// TIA Portal V15.1 export
// export: Created 2024-06-21T08:41:25.0501591Z, ExportSetting WithDefaults, DisplayName Totally Integrated Automation Portal, DisplayVersion V15.1 Update 5, DisplayName TIA Portal Openness, DisplayVersion V15.1 Update 5, DisplayName SINAMICS Startdrive Advanced, DisplayVersion V15.1, DisplayName G130, G150, S120, S150, SINAMICS MV, S210, DisplayVersion V15.1, DisplayName G110M, G120, G120C, G120D, G120P, DisplayVersion V15.1, DisplayName STEP 7 Professional, DisplayVersion V15.1 Update 5, DisplayName STEP 7 Safety, DisplayVersion V15.1, DisplayName WinCC Professional, DisplayVersion V15.1 Update 5, DisplayName SIMATIC Visualization Architect, DisplayVersion V15.1
FUNCTION_BLOCK "209230NCB01TagSeq"   // FB440, GRAPH
{ S7_Optimized_Access := 'TRUE' }
VERSION : 0.1
// stored: AcknowledgeErrorsRequired true, AutoNumber false, GraphVersion 6.0, InitialValuesAcquisition false, IsIECCheckEnabled false, LanguageInNetworks FBD, LockOperatingMode false, PermanentILProcessingInMANMode false, SetENOAutomatically false, SkipSteps false, UDAEnableTagReadback false, WithAlarmHandling true
   // inherited from GRAPH_BASE
   VAR
      OFF_SQ_BASE : Bool;
   END_VAR
   VAR_INPUT
      OFF_SQ { ExternalWritable := 'False'} : Bool := false;   // Turn sequence off
      INIT_SQ { ExternalWritable := 'False'} : Bool := false;   // Set sequence to initial state
      ACK_EF { ExternalWritable := 'False'} : Bool := false;   // Acknowledge all errors and faults
      S_PREV { ExternalWritable := 'False'} : Bool := false;   // Output previous step in parameter S_NO
      S_NEXT { ExternalWritable := 'False'} : Bool := false;   // Indicate next step in parameter S_NO
      SW_AUTO { ExternalWritable := 'False'} : Bool := false;   // Automatic mode
      SW_TAP { ExternalWritable := 'False'} : Bool := false;   // Semiautomatic/switch with transition
      SW_TOP { ExternalWritable := 'False'} : Bool := false;   // Semiautomatic/ignore transition
      SW_MAN { ExternalWritable := 'False'} : Bool := false;   // Manual mode
      S_SEL { ExternalWritable := 'False'} : Int := 0;   // Select step to be output to S_NO
      S_ON { ExternalWritable := 'False'} : Bool := false;   // Activate step indicated in S_NO
      S_OFF { ExternalWritable := 'False'} : Bool := false;   // Deactivate step indicated S_NO
      T_PUSH { ExternalWritable := 'False'} : Bool := false;   // Enable transition to switch in semi automatic mode
   END_VAR
   VAR_OUTPUT
      S_NO { ExternalWritable := 'False'} : Int := 0;   // Step number
      S_MORE { ExternalWritable := 'False'} : Bool := false;   // More steps are available and can be shown in S_NO
      S_ACTIVE { ExternalWritable := 'False'} : Bool := false;   // Step indicated in S_NO is active
      ERR_FLT { ExternalWritable := 'False'} : Bool := false;   // Interlock or supervision group error
      AUTO_ON { ExternalWritable := 'False'} : Bool := false;   // Automatic mode is active
      TAP_ON { ExternalWritable := 'False'} : Bool := false;   // Semiautomatic mode/step with transition enabled
      TOP_ON { ExternalWritable := 'False'} : Bool := false;   // Semiautomatic mode/ignore transition enabled
      MAN_ON { ExternalWritable := 'False'} : Bool := false;   // Manual mode is active
   END_VAR
BEGIN
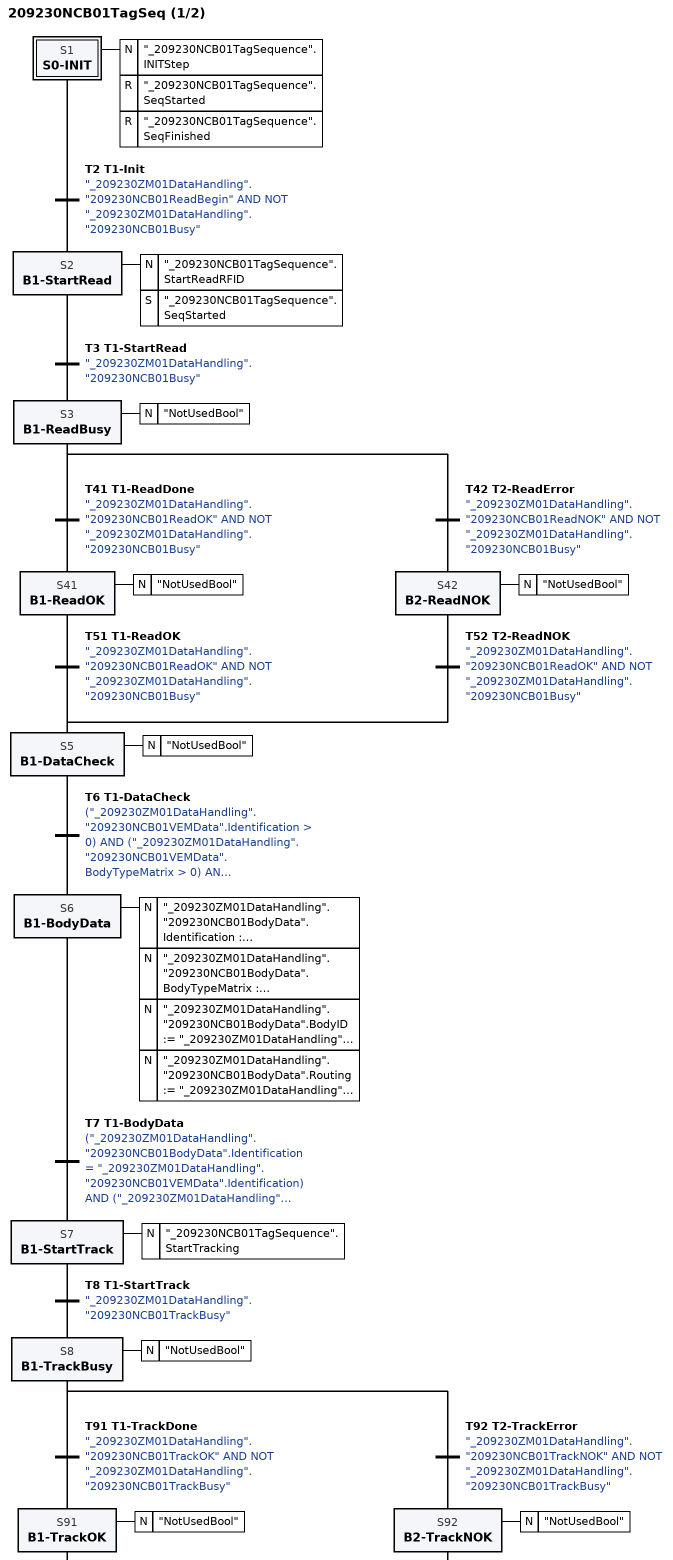
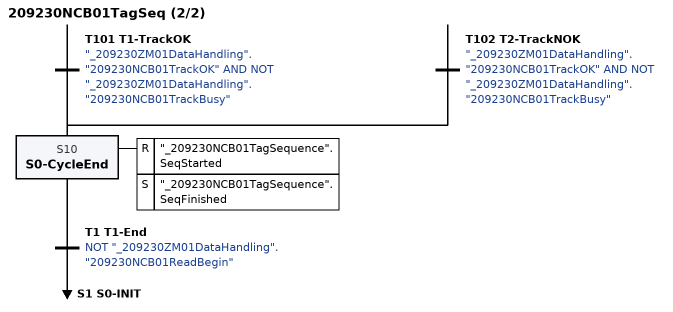
   // sequencer 1: 209230NCB01 Tag Sequence
   // Tag Sequence of 209230NCB01
   INITIAL_STEP "S0-INIT":   // S1, max time T#10S, warning time T#7S
      interlock C := (none);   // Not used
      supervision V := (none);   // Not Used
      // INIT
              N    "_209230NCB01TagSequence".INITStep
              R    "_209230NCB01TagSequence".SeqStarted
              R    "_209230NCB01TagSequence".SeqFinished
   END_STEP
   TRANSITION "T1-Init" FROM "S0-INIT" TO "B1-StartRead"   // T2
      := "_209230ZM01DataHandling"."209230NCB01ReadBegin" AND NOT "_209230ZM01DataHandling"."209230NCB01Busy";
   END_TRANSITION
   STEP "B1-StartRead":   // S2, max time T#10S, warning time T#7S
      interlock C := (none);   // Not Used
      supervision V := (none);   // Not Used
      // Start Getting VEM Data by Reading the Tag with RFID
              N    "_209230NCB01TagSequence".StartReadRFID
              S    "_209230NCB01TagSequence".SeqStarted
   END_STEP
   TRANSITION "T1-StartRead" FROM "B1-StartRead" TO "B1-ReadBusy"   // T3
      := "_209230ZM01DataHandling"."209230NCB01Busy";
   END_TRANSITION
   STEP "B1-ReadBusy":   // S3, max time T#10S, warning time T#7S
      interlock C := (none);   // Not Used
      supervision V := (none);   // Not Used
      // The Tag Reading is Busy
              N    "NotUsedBool"
   END_STEP
   TRANSITION "T1-ReadDone" FROM "B1-ReadBusy" TO "B1-ReadOK"   // T41
      := "_209230ZM01DataHandling"."209230NCB01ReadOK" AND NOT "_209230ZM01DataHandling"."209230NCB01Busy";
   END_TRANSITION
   TRANSITION "T2-ReadError" FROM "B1-ReadBusy" TO "B2-ReadNOK"   // T42
      := "_209230ZM01DataHandling"."209230NCB01ReadNOK" AND NOT "_209230ZM01DataHandling"."209230NCB01Busy";
   END_TRANSITION
   STEP "B1-ReadOK":   // S41, max time T#10S, warning time T#7S
      interlock C := (none);   // Not Used
      supervision V := (none);   // Not Used
      // Reading of Tag is OK
              N    "NotUsedBool"
   END_STEP
   TRANSITION "T1-ReadOK" FROM "B1-ReadOK" TO "B1-DataCheck"   // T51
      := "_209230ZM01DataHandling"."209230NCB01ReadOK" AND NOT "_209230ZM01DataHandling"."209230NCB01Busy";
   END_TRANSITION
   STEP "B2-ReadNOK":   // S42, max time T#10S, warning time T#7S
      interlock C := (none);   // Not Used
      supervision V := (none);   // Not Used
      // Reading of Tag is Not OK
              N    "NotUsedBool"
   END_STEP
   TRANSITION "T2-ReadNOK" FROM "B2-ReadNOK" TO "B1-DataCheck"   // T52
      := "_209230ZM01DataHandling"."209230NCB01ReadOK" AND NOT "_209230ZM01DataHandling"."209230NCB01Busy";
   END_TRANSITION
   STEP "S0-CycleEnd":   // S10, max time T#10S, warning time T#7S
      interlock C := (none);   // Not Used
      supervision V := (none);   // Not Used
      // Finished
              R    "_209230NCB01TagSequence".SeqStarted
              S    "_209230NCB01TagSequence".SeqFinished
   END_STEP
   TRANSITION "T1-End" FROM "S0-CycleEnd" TO "S0-INIT"   // T1, jump
      := NOT "_209230ZM01DataHandling"."209230NCB01ReadBegin";
   END_TRANSITION
   STEP "B1-DataCheck":   // S5, max time T#10S, warning time T#7S
      interlock C := (none);   // Not Used
      supervision V := (none);   // Not Used
      // Check if the Received Data is Valid
              N    "NotUsedBool"
   END_STEP
   TRANSITION "T1-DataCheck" FROM "B1-DataCheck" TO "B1-BodyData"   // T6
      := ("_209230ZM01DataHandling"."209230NCB01VEMData".Identification > 0) AND ("_209230ZM01DataHandling"."209230NCB01VEMData".BodyTypeMatrix > 0) AND ("_209230ZM01DataHandling"."209230NCB01VEMData".BodyID > 0) AND ("_209230ZM01DataHandling"."209230NCB01VEMData".BodyID <= 9999999) AND "_209230ZM01DataHandling"."209230NCB01VEMDataValid";
   END_TRANSITION
   STEP "B1-BodyData":   // S6, max time T#10S, warning time T#7S
      interlock C := (none);   // Not Used
      supervision V := (none);   // Not Used
      // Prepare Data for local use (ex. Shift Register)
              N    "_209230ZM01DataHandling"."209230NCB01BodyData".Identification := "_209230ZM01DataHandling"."209230NCB01VEMData".Identification
              N    "_209230ZM01DataHandling"."209230NCB01BodyData".BodyTypeMatrix := "_209230ZM01DataHandling"."209230NCB01VEMData".BodyTypeMatrix
              N    "_209230ZM01DataHandling"."209230NCB01BodyData".BodyID := "_209230ZM01DataHandling"."209230NCB01VEMData".BodyID
              N    "_209230ZM01DataHandling"."209230NCB01BodyData".Routing := "_209230ZM01DataHandling"."209230NCB01VEMData".Routing
   END_STEP
   TRANSITION "T1-BodyData" FROM "B1-BodyData" TO "B1-StartTrack"   // T7
      := ("_209230ZM01DataHandling"."209230NCB01BodyData".Identification = "_209230ZM01DataHandling"."209230NCB01VEMData".Identification) AND ("_209230ZM01DataHandling"."209230NCB01BodyData".BodyTypeMatrix = "_209230ZM01DataHandling"."209230NCB01VEMData".BodyTypeMatrix) AND ("_209230ZM01DataHandling"."209230NCB01BodyData".BodyID = "_209230ZM01DataHandling"."209230NCB01VEMData".BodyID) AND ("_209230ZM01DataHandling"."209230NCB01BodyData".Routing = "_209230ZM01DataHandling"."209230NCB01VEMData".Routing);
   END_TRANSITION
   STEP "B1-StartTrack":   // S7, max time T#10S, warning time T#7S
      interlock C := (none);   // Not Used
      supervision V := (none);   // Not Used
      // Start Tracking the Body
              N    "_209230NCB01TagSequence".StartTracking
   END_STEP
   TRANSITION "T1-StartTrack" FROM "B1-StartTrack" TO "B1-TrackBusy"   // T8
      := "_209230ZM01DataHandling"."209230NCB01TrackBusy";
   END_TRANSITION
   STEP "B1-TrackOK":   // S91, max time T#10S, warning time T#7S
      interlock C := (none);   // Not Used
      supervision V := (none);   // Not Used
      // Tracking of the Body is OK
              N    "NotUsedBool"
   END_STEP
   TRANSITION "T1-TrackOK" FROM "B1-TrackOK" TO "S0-CycleEnd"   // T101
      := "_209230ZM01DataHandling"."209230NCB01TrackOK" AND NOT "_209230ZM01DataHandling"."209230NCB01TrackBusy";
   END_TRANSITION
   STEP "B2-TrackNOK":   // S92, max time T#10S, warning time T#7S
      interlock C := (none);   // Not Used
      supervision V := (none);   // Not Used
      // Tracking of the Body is Not OK
              N    "NotUsedBool"
   END_STEP
   TRANSITION "T2-TrackNOK" FROM "B2-TrackNOK" TO "S0-CycleEnd"   // T102
      := "_209230ZM01DataHandling"."209230NCB01TrackOK" AND NOT "_209230ZM01DataHandling"."209230NCB01TrackBusy";
   END_TRANSITION
   STEP "B1-TrackBusy":   // S8, max time T#10S, warning time T#7S
      interlock C := (none);   // Not Used
      supervision V := (none);   // Not Used
      // The Body Tracking is Busy
              N    "NotUsedBool"
   END_STEP
   TRANSITION "T1-TrackDone" FROM "B1-TrackBusy" TO "B1-TrackOK"   // T91
      := "_209230ZM01DataHandling"."209230NCB01TrackOK" AND NOT "_209230ZM01DataHandling"."209230NCB01TrackBusy";
   END_TRANSITION
   TRANSITION "T2-TrackError" FROM "B1-TrackBusy" TO "B2-TrackNOK"   // T92
      := "_209230ZM01DataHandling"."209230NCB01TrackNOK" AND NOT "_209230ZM01DataHandling"."209230NCB01TrackBusy";
   END_TRANSITION

   // permanent post-instructions: Not Used
END_FUNCTION_BLOCK
